	DATA_BLOCK DB161
	TITLE =DBG061M  AERATION AIR STEEPING 15
	//COPYRIGHT:    (C) 2009  BUHLER AG, CH-9240 UZWIL, SWITZERLAND
	//
	//PRODUCT:      WinCoS_BIW01_09
	//
	//TITLE:        AERATION AIR STEEPING 15
	//                Machine group DB
	//                Maschinengruppen-DB
	//
	//-------------------------------------------------------------------------
	//
	//IDENT:        AUTHOR:             DEPT:             DATE:
	//
	//P01_DB161.1.0 K.Renz              CSB41             13.Jan.2010
	//              1st Release
	//
	//-------------------------------------------------------------------------
	//
	//PURPOSE:
	//
	//MANUAL :
	//
	//RESTRICTIONS:
	//
	//-------------------------------------------------------------------------
	AUTHOR  : KR
	FAMILY  : USW
	NAME    : DBG061M
	VERSION : 00.00

	FB161
	BEGIN
	      #Gr.Par.ParObjectNo 	:=6100;
	      #Gr.Par.ParIdling      	:=2;
	      #Gr.Par.ParMgr	        :=True;
	      #Gr.Par.ParWgr	        :=False;
	      #Gr.Par.ParGgr	        :=False;
	      #Gr.Par.ParEmptyingTime 	:=0;
	      #Gr.Par.ParHornCode       :=1;
	//Parameter =A-1125-QXV/BZS41/42 : AERATION AIR RING ST 15
	      #A_1125_QXV_BZS41_42.Par.ParObjectNo                             :=6101;
	      #A_1125_QXV_BZS41_42.Par.ParMsgType                              :=7081;
	      #A_1125_QXV_BZS41_42.Par.ParHornCode                             :=1;
	      #A_1125_QXV_BZS41_42.Par.ParMonTime                              :=100;
	      #A_1125_QXV_BZS41_42.Par.ParPulseTimeHN                          :=5;
	      #A_1125_QXV_BZS41_42.Par.ParPulseTimeLN                          :=5;
	      #A_1125_QXV_BZS41_42.Par.ParIdlingTime                           :=0;
	      #A_1125_QXV_BZS41_42.Par.ParDelayTime                            :=0;
	      #A_1125_QXV_BZS41_42.Par.ParLogOff                               :=False;
	      #A_1125_QXV_BZS41_42.Par.ParManual                               :=True;
	      #A_1125_QXV_BZS41_42.Par.ParPulseValve                           :=False;
	      #A_1125_QXV_BZS41_42.Par.ParContValve                            :=True;
	      #A_1125_QXV_BZS41_42.Par.ParManualFlap                           :=False;
	//
	//
	END_DATA_BLOCK
